FUNCTION_BLOCK TcoStateAutoRestoreTest EXTENDS TcoState
VAR
    _myState : INT;
    _onStateChangeCounter : INT;
    _restoreCounter : INT;
    _autoRestoreToMyChildsEnabled : BOOL;
    _autoRestoreByMyParentEnabled : BOOL;
    _countsPerStep : ULINT;
    _counterValue : ULINT;
END_VAR

{attribute 'TcRpcEnable'}
METHOD INTERNAL CleanUp
THIS^.ChangeState(0);
_myState := State;
_onStateChangeCounter := 0;
_restoreCounter := 0;
_autoRestoreToMyChildsEnabled := FALSE;
_autoRestoreByMyParentEnabled := FALSE;
_countsPerStep := 0;
_counterValue := 0;
END_METHOD

{attribute 'TcRpcEnable'}
METHOD INTERNAL ExecutionBody
IF State = -1 THEN
    _counterValue := 0;
    ChangeState(0);
END_IF

IF State = 0 THEN
    _counterValue := _counterValue + 1;

    IF (_counterValue MOD _countsPerStep) = 0 THEN
        ChangeState(State + 10);
    END_IF
END_IF

IF State = 10 THEN
    _counterValue := _counterValue + 1;

    IF (_counterValue MOD _countsPerStep) = 0 THEN
        ChangeState(State + 10);
    END_IF
END_IF

IF State = 20 THEN
    _counterValue := _counterValue + 1;

    IF (_counterValue MOD _countsPerStep) = 0 THEN
        ChangeState(State + 10);
    END_IF
END_IF

IF State = 30 THEN
    _counterValue := _counterValue + 1;

    IF (_counterValue MOD _countsPerStep) = 0 THEN
        ChangeState(State + 10);
    END_IF
END_IF

IF State = 40 THEN
    _counterValue := _counterValue + 1;

    IF (_counterValue MOD _countsPerStep) = 0 THEN
        ChangeState(State + 10);
    END_IF
END_IF

IF State = 50 THEN
    _counterValue := _counterValue + 1;

    IF (_counterValue MOD _countsPerStep) = 0 THEN
        ChangeState(State + 10);
    END_IF
END_IF

IF State = 60 THEN
    ChangeState(-1);
END_IF

_myState := State;
END_METHOD

METHOD PROTECTED OnStateChange
VAR_INPUT
    PreviousState : INT;
    NewState : INT;
END_VAR
_onStateChangeCounter := _onStateChangeCounter + 1;
SUPER^.OnStateChange(PreviousState, NewState);
END_METHOD

{attribute 'TcRpcEnable'}
METHOD INTERNAL ReadOutAutoRestoreProperties
_autoRestoreToMyChildsEnabled := THIS^.IsAutoRestoreEnabled;
_autoRestoreByMyParentEnabled := THIS^.AutoRestorable;
END_METHOD

METHOD Restore : ITcoRestorable
_restoreCounter := _restoreCounter + 1;
SUPER^.Restore();
END_METHOD

{attribute 'TcRpcEnable'}
METHOD INTERNAL TriggerRestore
THIS^.Restore();
_myState := State;
END_METHOD

END_FUNCTION_BLOCK

(* stored: Version 1.1.0.1
   POU TcoStateAutoRestoreTest: Id {635180e2-b2d9-4213-a2a6-8bd32b517b3b}, SpecialFunc None
   Method CleanUp: Id {081b5928-de47-4761-be4d-83ea89a64bf4}
   Method ExecutionBody: Id {680585de-c3db-4af0-b280-e5ea8b43e2b4}
   Method OnStateChange: Id {de76d52f-5157-49e1-8531-4b05abb17ada}
   Method ReadOutAutoRestoreProperties: Id {fa3f5405-9438-4099-9edf-95c6d9998cd8}
   Method Restore: Id {8a149d97-03d1-42be-b1ec-fe88428a36b7}
   Method TriggerRestore: Id {c5028e48-ff1c-497f-9f19-1a366dc1e69a} *)
